// TIA Portal V19 export
VAR_GLOBAL   // PLC tag table "CoilCar_IO"
   Coilcar_Lift1_Ls_Down AT %I128.5 : Bool;   // 796SQ1
   Coilcar_Lift1_Ls_Up AT %I128.6 : Bool;   // 796SQ2
   Coilcar_Lift1_V_Down AT %Q102.7 : Bool;   // 796YV1
   Coilcar_Lift1_V_Up AT %Q103.0 : Bool;   // 796YV2
   Coilcar_Lift2_Ls_Down AT %I128.7 : Bool;   // 797SQ1
   Coilcar_Lift2_Ls_Up AT %I129.0 : Bool;   // 797SQ2
   Coilcar_Lift2_V_Down AT %Q103.1 : Bool;   // 797YV1
   Coilcar_Lift2_V_Up AT %Q103.2 : Bool;   // 797YV2
   Culla_Controllo_Perni_Inseriti_Phc_1 AT %I127.4 : Bool;   // 788BF1
   Culla_Controllo_Perni_Inseriti_Phc_2 AT %I127.5 : Bool;   // 788BF2
   Culla_Controllo_Perni_Inseriti_Phc_3 AT %I127.6 : Bool;   // 788BF3
   Culla_Controllo_Perni_Inseriti_Phc_4 AT %I127.7 : Bool;   // 788BF4
   Culla_Ls_Indietro_Minimo_Fuori_Linea AT %I128.0 : Bool;   // 795SQ1
   Culla_Ls_Avanti_Massimo_In_Linea AT %I128.1 : Bool;   // 795SQ2
   Culla_Ls_Rallentamento_Indietro AT %I128.2 : Bool;   // 795SQ3
   Culla_Ls_Rallentamento_Avanti AT %I128.3 : Bool;   // 795SQ4
   Culla_Ls_Coil_Inserito_Togliere_Perni AT %I128.4 : Bool;   // 795SQ5
END_VAR
